(* PLC project Tc2_Utilities.UInt64Min Demo, tc3-libraries-kb TwinCAT 3.1 *)
(* stored: creationDateTime 2026-05-12T12:00:00, modificationDateTime 2026-05-12T12:00:00 *)

PROGRAM P_Demo_UInt64Min
  VAR
    uliLineA : T_ULARGE_INTEGER;;  (* A 线剩余 *)
    uliLineB : T_ULARGE_INTEGER;;  (* B 线剩余 *)
    uliMin : T_ULARGE_INTEGER;;  (* 瓶颈 *)
    bPick : BOOL;
  END_VAR

            // ============================================================
// Tc2_Utilities.UInt64Min 演示程序（FUNCTION，单周期触发）
// ============================================================
// 场景：选定两个生产线的剩余容量中较小者作为系统瓶颈。
// 价值：替代手写 IF/ELSE；一次调用。
// 验证步骤：
//   1. 把本 PROGRAM 加到 PlcTask 调用列表
//   2. 编译 + 登录
//   3. 在线把 b... 触发位置 TRUE 一个周期
//   4. 观察输出变量是否符合期望
// ============================================================

IF bPick THEN
    uliMin := UInt64Min(uliLineA, uliLineB);
    bPick := FALSE;
END_IF;

          
END_PROGRAM
